TYPE LG_set :
STRUCT
	Coils	:	LG_Coils;
	Regs	:	LG_ControlRegs;
END_STRUCT
END_TYPE

(* stored: Version 1.1.0.1, ProductVersion 3.1.4024.12
   DUT LG_set: Id {238bd9ff-acc1-4c57-ab1d-1d4693b7210d} *)
